//EL7211 | Servo terminal, for resolver, 50V DC, 4.5Arms
FUNCTION_BLOCK EL7211

VAR_INPUT
	En: BOOL;
	iTerminal_ID : INT;
	ErrorSystem : POINTER TO ST_ErrorSystem;
END_VAR

VAR_OUTPUT
	EnO: BOOL;
	bError: BOOL;
END_VAR

VAR
	//WC_State is handled by NC, so NOT included here.
	InfoData_State AT %I*: UINT;
	
	//FB-s
	EL7211_Error 	: FB_TerminalError;
END_VAR

(*
* TODO: Test on hardware
*)

EnO:=En;

EL7211_Error(
	En := TRUE,
	iTerminal_ID := iTerminal_ID,
	bWcState := FALSE,
	uiInfoData_State := InfoData_State,
	pErrorSystem := ErrorSystem,
	bError => bError,
);

END_FUNCTION_BLOCK

(* stored: Version 1.1.0.1, ProductVersion 3.1.4022.17
   POU EL7211: Id {b42893c3-600d-478d-8498-9389d8fa4a5c}, SpecialFunc None *)
